FUNCTION_BLOCK FB_ArrayDint VAR_GENERIC CONSTANT nLength: DINT:= 1; END_VAR
VAR_INPUT
END_VAR
VAR_OUTPUT
END_VAR
VAR
	nValues:			ARRAY [0..nLength - 1] OF DINT;
END_VAR

END_FUNCTION_BLOCK

(* stored: Version 1.1.0.1
   POU FB_ArrayDint: Id {1b6e5608-6533-03be-0953-370b0ccf8f1c}, SpecialFunc None *)
